{attribute 'qualified_only'}
VAR_GLOBAL
	
	PowerOn:				BOOL;
	MotionPowerOn:			BOOL;

	PowerOnFdbk:			BOOL; //power feedback
	MotionPowerOnFdbk:		BOOL; //power feedback

 	Data: typeStationMode;
	
	//all Unit rows in the station, to be used as the "Mc" station
	UnitRow: ARRAY[1..99] OF typeMotionRow;
	UnitRowBtn: ARRAY[1..99] OF typeMotionRowButtons;

END_VAR

(* stored: Version 1.1.0.1, ProductVersion 3.1.4024.12
   GVL Mc_Global: Id {5642ad69-83f7-4656-9927-4be704aafe8e} *)
